Staubli VAL3: onF2Event.pgx

program onF2Event()
  local tool l_tTool
  local bool l_bContinue
  local num i
  local num l_nSize
begin
  // look if the bButton is enable
  if bButton[1]
    if cycleStatus:bSimulation
      //
      // ENABLE STEPPING
      //
      call trajType:getSizeItem(false,l_nSize)
      if !bStepping and nPoint<(l_nSize-1) and taskStatus("stepping")==-1 and !isEmpty()
        taskCreate "stepping",20,stepping()
      endIf
    else
      //
      // go to actual POINT
      //
      if !cycleStatus:bCycle or !cycleStatus:bSimulation
        call goTo(nPoint)
      endIf
    endIf
  endIf
end
